FUNCTION_BLOCK FB_Cinta EXTENDS FB_Module
VAR_INPUT
	Situar: BOOL;
	Transferir: BOOL;
	
	TE: TIME := T#0.5S;
	TR: TIME := T#0.5S;
	TS: TIME := T#0.5S;
	TT: TIME := T#1S;
	TX: TIME := T#1S;
END_VAR
VAR
	fbController: FB_Cinta_SFC;

	(* Sensores especificos *)
	pp: dvSensor; // presencia de pale

	(* Actuadores especificos *)
	RUN: dvActuator; // activa motor
	REV: dvActuator; // invierte motor
	R_1: dvActuator; // retenedor baja
	S_1: dvActuator; // separador sube
END_VAR

METHOD InitialConditions : BOOL
VAR_INPUT
END_VAR
InitialConditions:= TRUE;
END_METHOD

METHOD ModuleControlFlow : BOOL


fbController.SFCPause := Pausar;
fbController.SFCReset := Reset;

pp.ProcessCycle(gm.ModeActual, sfcValue=>fbController.pp);
IC := InitialConditions();

fbController(	
	tm := tm, IC:=IC, Execute:=Execute, Ack:=Ack,
	Situar := Situar, Transferir := Transferir,
	Ready=>Ready, Done=>Done, Failure=>Failure);

RUN.ProcessCycle(gm.ModeActual, sfcValue:=fbController.RUN);
REV.ProcessCycle(gm.ModeActual, sfcValue:=fbController.REV);
R_1.ProcessCycle(gm.ModeActual, sfcValue:=fbController.R_1);
S_1.ProcessCycle(gm.ModeActual, sfcValue:=fbController.S_1);
END_METHOD

END_FUNCTION_BLOCK

(* stored: Version 1.1.0.1, ProductVersion 3.1.4024.6
   POU FB_Cinta: Id {f4de692b-96c6-493e-9b33-3a90e20acfad}, SpecialFunc None
   Method InitialConditions: Id {6207c809-4e5c-471b-9748-498f300af54e}
   Method ModuleControlFlow: Id {8ef223d1-a933-4fe3-87e8-40d9ed750433} *)
